Yaskawa INFORM job: R1_TOOLPOUNCE_BLK.JBI

/JOB
//NAME R1_TOOLPOUNCE_BLK
//POS
///NPOS 0,0,0,0,0,0
//INST
///DATE 2021/09/30 10:12
///ATTR SC,RW
///GROUP1 RB1
///LVARS 0,0,0,0,0,0,0,0
NOP
'%%%%%%%%%%%%%%%%%%%%%%%%%%%%%%%%
' R1 Tool Change Pounce Position
'%%%%%%%%%%%%%%%%%%%%%%%%%%%%%%%%
'
*TOP
'***********INITIALIZE***********
'********************************
'
'********PRE-STATUS_CHECK********
' Set Clear of Module Bits
CALL JOB:R1_CLEARMODULE ARGF242
' Report Position
CALL JOB:R1_REPORTPOS ARGF10
'********************************
'
'***********PRIME_MOVE***********
'********************************
IFTHENEXP B005=0
	 MOVJ P[106] VJ=25.00
ENDIF
'
'*******POST-STATUS_CHECK********
'********************************
'
'****USER_DEFINED_PARAMETERS*****
'********************************
'
'********DATA_VALIDATION*********
'********************************
'
'*************SETUP**************
'********************************
'
'*************ACTION*************
'********************************
'
'*********HOUSE_KEEPING**********
SET B004 1
'********************************
*OUT
END
